{attribute addProperty BoxType "EL4031-0000-0016"}
{attribute addProperty Id "AO_OutputsAT %Q*AO_Outputs_F57FA4F91620WcStateAT %I*WcState_28A8677510.1250InfoDataAT %I*InfoData_BC63D37F80100"}
{attribute addProperty CRC "1097990690"}
{attribute addProperty SizeInBites "97"}
{attribute addProperty SizeInBytes "12.125"}
TYPE EL4031_50B5189C :
STRUCT
	{attribute addProperty Name "AO_Outputs"}
	AO_Outputs : AO_Outputs_F57FA4F9;
	{attribute addProperty Name "WcState"}
	WcState : WcState_28A86775;
	{attribute addProperty Name "InfoData"}
	InfoData : InfoData_BC63D37F;
END_STRUCT
END_TYPE

(* stored: Version 1.2.0.0, ProductVersion 3.1.4024.9
   DUT EL4031_50B5189C: Id {d7b932b9-58d8-490e-b6c4-321c581de097} *)
